Staubli VAL3: readSocket.pgx

program readSocket(num x_nCamID (dimensions=1), string& x_sMsg[] (dimensions=1), bool& x_bError[] (dimensions=1))
  local num l_nChar
  local num l_nCount
begin
  //-----------------------------------------------------------------------
  //Header begin
  //Description of program
  //  Read string from socket.
  //
  //Input parameters
  //  num x_nCamID :
  //    role : camera's ID
  //
  //Output parameters
  //  string x_sMsg :
  //    role : native command
  //  bool x_bError :
  //    role : returns true if an error occurred and false otherwise
  //
  //Examples
  //  call readSocket(nCamID,l_sMsgError,l_bError)
  //
  //
  //  Creation : 19-05-08 - f.Rob
  //Header end
  //-----------------------------------------------------------------------

  x_sMsg=""
  do
    l_nCount=sioGet(cCamera[x_nCamID].sSocket,l_nChar)
    //-1 : timeout for input communication has been reached
    if (l_nCount>-1) and (l_nChar>=32)
      x_sMsg=x_sMsg+chr(l_nChar)
    endIf
    x_bError=l_nCount<=-1
  until (l_nChar==13) or x_bError
  //Displays error message
  if bDebugSocket
    ? "R Status code> "+x_sMsg
  endIf
end
